// TIA Portal V17 export
// export: Created 2022-07-20T06:59:51.9374279Z, ExportSetting WithDefaults, DisplayName Totally Integrated Automation Portal, DisplayVersion V17, DisplayName TIA Portal Openness, DisplayVersion V17, DisplayName TIA Portal Version Control Interface, DisplayVersion V17, DisplayName SINAMICS Startdrive Advanced, DisplayVersion V17, DisplayName SINAMICS Startdrive G130, G150, S120, S150, SINAMICS MV, S210, DisplayVersion V17, DisplayName SINAMICS Startdrive G110M, G120, G120C, G120D, G120P, G115D, DisplayVersion V17, DisplayName STEP 7 Professional, DisplayVersion V17, DisplayName STEP 7 Safety, DisplayVersion V17, DisplayName WinCC Advanced, DisplayVersion V17
FUNCTION_BLOCK "FB10080_UvLedsManager"   // FB10080, LAD
{ S7_Optimized_Access := 'TRUE' }
VERSION : 0.1
// stored: AutoNumber false, IsIECCheckEnabled false, IsRetainMemResEnabled false, MemoryReserve 100, SetENOAutomatically false, UDAEnableTagReadback false
   VAR_INPUT
      UvLedsSetPoint : Real;   // 0..100%
      RequestUvLedsActivation : Bool;
   END_VAR
   VAR_OUTPUT
      ActiveUvLeds : Bool;
      AnalogicalPowerValue : Real;
      UvLedsActivated : Bool;
   END_VAR
   VAR
      TON_SafetyUvLeds : TON_TIME;
   END_VAR
BEGIN

REGION Network 1 (SCL): First Scan
   IF "FirstScan" THEN
       #ActiveUvLeds := FALSE;
       #AnalogicalPowerValue := 0.0;
   END_IF;
END_REGION

REGION Network 2 (SCL): Edge Signals & Timers
   REGION EDGE SIGNALS
   END_REGION

   REGION TIMERS
       #TON_SafetyUvLeds(IN := #ActiveUvLeds,
                         PT := T#10s);
   END_REGION
END_REGION

REGION Network 3 (SCL): Uv Leds Management
   IF #RequestUvLedsActivation THEN
       #ActiveUvLeds := TRUE;
       "FC10010_ScalingPercentageToAnalog"(SetPoint := #UvLedsSetPoint,
                                           AnalogValue => #AnalogicalPowerValue);
       #UvLedsActivated := TRUE;
   ELSE
       #ActiveUvLeds := FALSE;
       #AnalogicalPowerValue := 0.0;
       #UvLedsActivated := FALSE;
   END_IF;
END_REGION

REGION Network 4 (SCL): Safety Management
END_REGION
END_FUNCTION_BLOCK
